Omron CX-Programmer project NewProject (CX-Programmer 9.73)

# PLC NewPLC1: CP1E E20

## Global symbols (name address type ; comment)
0 CHANNEL  ; TIMPROS1
0.00 BOOL  ; NO1
0.03 BOOL  ; NO2
0.08 BOOL  ; A1
0.09 BOOL  ; A2
0.10 BOOL  ; A3
1.00 BOOL  ; ON
1.04 BOOL  ; NO3
2.00 BOOL  ; OFF
2.01 BOOL  ; OFF
2.02 BOOL  ; NC1
3.00 BOOL  ; NC2
3.03 BOOL  ; PROSES1
3.05 BOOL  ; NC2
4.00 BOOL  ; NC3
4.06 BOOL  ; NC3
5.00 BOOL  ; NC4
5.07 BOOL  ; NC4
6.00 BOOL  ; CONVE
6.02 BOOL  ; CONVEYOR
T000 BOOL  ; T1
T001 BOOL  ; T2
T002 BOOL  ; T3

## Program NewProgram1 (cyclic task 0)
; KONVEYTUGAS
Local symbols
TIM 0.00 BOOL

### Section Section1
; TUGAS INI BANG

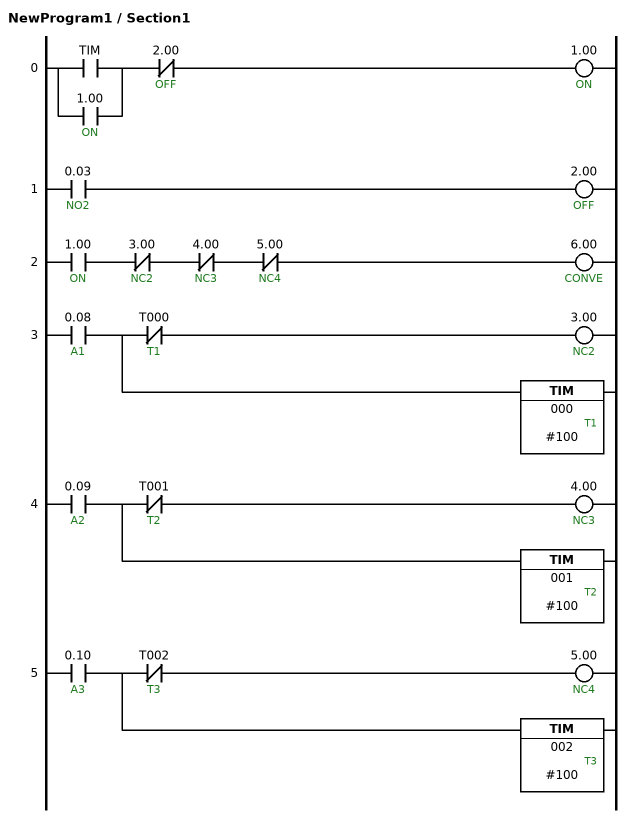
; rung 0
LD TIM
OR 1.00  ; ON
ANDNOT 2.00  ; OFF
OUT 1.00  ; ON
; rung 1
LD 0.03  ; NO2
OUT 2.00  ; OFF
; rung 2
LD 1.00  ; ON
ANDNOT 3.00  ; NC2
ANDNOT 4.00  ; NC3
ANDNOT 5.00  ; NC4
OUT 6.00  ; CONVE
; rung 3
LD 0.08  ; A1
OUT TR0
ANDNOT T000  ; T1
OUT 3.00  ; NC2
LD TR0
TIM 000 #100  ; T1
; rung 4
LD 0.09  ; A2
OUT TR0
ANDNOT T001  ; T2
OUT 4.00  ; NC3
LD TR0
TIM 001 #100  ; T2
; rung 5
LD 0.10  ; A3
OUT TR0
ANDNOT T002  ; T3
OUT 5.00  ; NC4
LD TR0
TIM 002 #100  ; T3

### Section END
; rung 0
END(001)